    car3/doorL2/doorControlPart/openedDoor AT 1085 : BOOL := false;
    car3/doorL2/doorControlPart/closedDoor AT 1086 : BOOL := false;
    car3/doorL2/doorControlPart/lockedDoor AT 1087 : BOOL := false;
    car3/doorL2/doorControlPart/unlockedDoor AT 1088 : BOOL := false;
    car3/doorL2/doorControlPart/openingRequest AT 1089 : BOOL := false;
    car3/doorL2/doorControlPart/doorOpeningCmd AT 1090 : BOOL := false;
    car3/doorL2/doorControlPart/doorClosingCmd AT 1091 : BOOL := false;
    car3/doorL2/doorControlPart/doorLockingCmd AT 1083 : BOOL := false;
    car3/doorL2/doorControlPart/doorUnlockingCmd AT 1084 : BOOL := false;
    car3/doorL2/doorControlPart/closedDoorState AT 38 : BOOL := false;
    car3/doorL2/doorControlPart/openedDoorState AT 37 : BOOL := false;
    car3/doorL2/doorControlPart/faultState AT 533 : DINT := 0;
    car3/doorL2/doorControlPart/_X_10 AT 1103 : BOOL := true;
    car3/doorL2/doorControlPart/_X_11 AT 1104 : BOOL := false;
    car3/doorL2/doorControlPart/_X_12 AT 1105 : BOOL := false;
    car3/doorL2/doorControlPart/_X_13 AT 1106 : BOOL := false;
    car3/doorL2/doorControlPart/_X_14 AT 1107 : BOOL := false;
    car3/doorL2/doorControlPart/_X_15 AT 1108 : BOOL := false;
    car3/doorL2/doorControlPart/_X_16 AT 1109 : BOOL := false;
    car3/doorL2/door/compressedAir AT 115 : REAL := 200.0;
    car3/doorL2/door/cmdSupply AT 1016 : BOOL := true;
    car3/doorL2/door/sensorSupply AT 1015 : BOOL := true;
    car3/doorL2/door/openDoorCmd AT 1090 : BOOL := false;
    car3/doorL2/door/closeDoorCmd AT 1091 : BOOL := false;
    car3/doorL2/door/lockActive AT 1092 : BOOL := false;
    car3/doorL2/door/doorOpened AT 1085 : BOOL := false;
    car3/doorL2/door/doorClosed AT 1086 : BOOL := false;
    car3/doorL2/door/increment AT 121 : REAL := 0.0;
    car3/doorL2/door/openDoor AT 1116 : BOOL := false;
    car3/doorL2/door/closeDoor AT 1117 : BOOL := false;
    car3/doorL2/door/doorPosition AT 122 : REAL := 0.0;
    car3/doorL2/door/length AT 123 : REAL := 1000.0;
    car3/doorL2/door/doorClosedSensorLogic AT 1118 : BOOL := true;
    car3/doorL2/door/doorOpenedSensorLogic AT 1119 : BOOL := true;
    car3/doorL2/door/d_locking AT 1120 : BOOL := false;
    car3/doorL2/door/v_d_locking AT 124 : REAL := 50.0;
    car3/doorL2/door/d_doorClosedSensor AT 1121 : BOOL := false;
    car3/doorL2/door/v_d_doorClosedSensor AT 1122 : BOOL := false;
    car3/doorL2/door/d_doorOpenedSensor AT 1123 : BOOL := false;
    car3/doorL2/door/v_d_doorOpenedSensor AT 1124 : BOOL := false;
    car3/doorL3/compressedAir AT 114 : REAL := 200.0;
    car3/doorL3/cmdSupply AT 1014 : BOOL := true;
    car3/doorL3/sensorSupply AT 1013 : BOOL := true;
    car3/doorL3/enableOpening AT 1019 : BOOL := false;
    car3/doorL3/enableClosing AT 1020 : BOOL := false;
    car3/doorL3/closedDoorState AT 36 : BOOL := false;
    car3/doorL3/openedDoorState AT 35 : BOOL := false;
    car3/doorL3/faultState AT 532 : DINT := 0;
    car3/doorL3/doorPB/doorPB AT 1131 : BOOL := false;
    car3/doorL3/doorPB/button AT 1135 : BOOL := false;
    car3/doorL3/doorPB/_X_10 AT 1136 : BOOL := true;
    car3/doorL3/doorPB/_X_11 AT 1137 : BOOL := false;
    car3/doorL3/doorPB/_X_12 AT 1138 : BOOL := false;
    car3/doorL3/doorLocking/lockingCmd AT 1125 : BOOL := false;
    car3/doorL3/doorLocking/unlockingCmd AT 1126 : BOOL := false;
    car3/doorL3/doorLocking/doorLocked AT 1129 : BOOL := false;
    car3/doorL3/doorLocking/doorUnlocked AT 1130 : BOOL := false;
    car3/doorL3/doorLocking/lockActive AT 1134 : BOOL := false;
    car3/doorL3/doorLocking/i_rs1 AT 662 : DINT := 0;
    car3/doorL3/doorLocking/d_unlockedSensor AT 1140 : BOOL := false;
    car3/doorL3/doorLocking/v_d_unlockedSensor AT 1141 : BOOL := false;
    car3/doorL3/doorLocking/d_lockedSensor AT 1142 : BOOL := false;
    car3/doorL3/doorLocking/v_d_lockedSensor AT 1143 : BOOL := false;
    car3/doorL3/doorControlPart/enableOpening AT 1019 : BOOL := false;
    car3/doorL3/doorControlPart/enableClosing AT 1020 : BOOL := false;
    car3/doorL3/doorControlPart/openedDoor AT 1127 : BOOL := false;
    car3/doorL3/doorControlPart/closedDoor AT 1128 : BOOL := false;
    car3/doorL3/doorControlPart/lockedDoor AT 1129 : BOOL := false;
    car3/doorL3/doorControlPart/unlockedDoor AT 1130 : BOOL := false;
    car3/doorL3/doorControlPart/openingRequest AT 1131 : BOOL := false;
    car3/doorL3/doorControlPart/doorOpeningCmd AT 1132 : BOOL := false;
    car3/doorL3/doorControlPart/doorClosingCmd AT 1133 : BOOL := false;
    car3/doorL3/doorControlPart/doorLockingCmd AT 1125 : BOOL := false;
    car3/doorL3/doorControlPart/doorUnlockingCmd AT 1126 : BOOL := false;
    car3/doorL3/doorControlPart/closedDoorState AT 36 : BOOL := false;
    car3/doorL3/doorControlPart/openedDoorState AT 35 : BOOL := false;
    car3/doorL3/doorControlPart/faultState AT 532 : DINT := 0;
    car3/doorL3/doorControlPart/_X_10 AT 1145 : BOOL := true;
    car3/doorL3/doorControlPart/_X_11 AT 1146 : BOOL := false;
    car3/doorL3/doorControlPart/_X_12 AT 1147 : BOOL := false;
    car3/doorL3/doorControlPart/_X_13 AT 1148 : BOOL := false;
    car3/doorL3/doorControlPart/_X_14 AT 1149 : BOOL := false;
    car3/doorL3/doorControlPart/_X_15 AT 1150 : BOOL := false;
    car3/doorL3/doorControlPart/_X_16 AT 1151 : BOOL := false;
    car3/doorL3/door/compressedAir AT 114 : REAL := 200.0;
    car3/doorL3/door/cmdSupply AT 1014 : BOOL := true;
    car3/doorL3/door/sensorSupply AT 1013 : BOOL := true;
    car3/doorL3/door/openDoorCmd AT 1132 : BOOL := false;
    car3/doorL3/door/closeDoorCmd AT 1133 : BOOL := false;
    car3/doorL3/door/lockActive AT 1134 : BOOL := false;
    car3/doorL3/door/doorOpened AT 1127 : BOOL := false;
    car3/doorL3/door/doorClosed AT 1128 : BOOL := false;
    car3/doorL3/door/increment AT 125 : REAL := 0.0;
    car3/doorL3/door/openDoor AT 1158 : BOOL := false;
    car3/doorL3/door/closeDoor AT 1159 : BOOL := false;
    car3/doorL3/door/doorPosition AT 126 : REAL := 0.0;
    car3/doorL3/door/length AT 127 : REAL := 1000.0;
    car3/doorL3/door/doorClosedSensorLogic AT 1160 : BOOL := true;
    car3/doorL3/door/doorOpenedSensorLogic AT 1161 : BOOL := true;
    car3/doorL3/door/d_locking AT 1162 : BOOL := false;
    car3/doorL3/door/v_d_locking AT 128 : REAL := 50.0;
    car3/doorL3/door/d_doorClosedSensor AT 1163 : BOOL := false;
    car3/doorL3/door/v_d_doorClosedSensor AT 1164 : BOOL := false;
    car3/doorL3/door/d_doorOpenedSensor AT 1165 : BOOL := false;
    car3/doorL3/door/v_d_doorOpenedSensor AT 1166 : BOOL := false;
    car3/doorR1/compressedAir AT 113 : REAL := 200.0;
    car3/doorR1/cmdSupply AT 1012 : BOOL := true;
    car3/doorR1/sensorSupply AT 1011 : BOOL := true;
    car3/doorR1/enableOpening AT 1021 : BOOL := false;
    car3/doorR1/enableClosing AT 1022 : BOOL := false;
    car3/doorR1/closedDoorState AT 34 : BOOL := false;
    car3/doorR1/openedDoorState AT 33 : BOOL := false;
    car3/doorR1/faultState AT 531 : DINT := 0;
    car3/doorR1/doorPB/doorPB AT 1173 : BOOL := false;
    car3/doorR1/doorPB/button AT 1177 : BOOL := false;
    car3/doorR1/doorPB/_X_10 AT 1178 : BOOL := true;
    car3/doorR1/doorPB/_X_11 AT 1179 : BOOL := false;
    car3/doorR1/doorPB/_X_12 AT 1180 : BOOL := false;
    car3/doorR1/doorLocking/lockingCmd AT 1167 : BOOL := false;
    car3/doorR1/doorLocking/unlockingCmd AT 1168 : BOOL := false;
    car3/doorR1/doorLocking/doorLocked AT 1171 : BOOL := false;
    car3/doorR1/doorLocking/doorUnlocked AT 1172 : BOOL := false;
    car3/doorR1/doorLocking/lockActive AT 1176 : BOOL := false;
    car3/doorR1/doorLocking/i_rs1 AT 665 : DINT := 0;
    car3/doorR1/doorLocking/d_unlockedSensor AT 1182 : BOOL := false;
    car3/doorR1/doorLocking/v_d_unlockedSensor AT 1183 : BOOL := false;
    car3/doorR1/doorLocking/d_lockedSensor AT 1184 : BOOL := false;
    car3/doorR1/doorLocking/v_d_lockedSensor AT 1185 : BOOL := false;
    car3/doorR1/doorControlPart/enableOpening AT 1021 : BOOL := false;
    car3/doorR1/doorControlPart/enableClosing AT 1022 : BOOL := false;
    car3/doorR1/doorControlPart/openedDoor AT 1169 : BOOL := false;
    car3/doorR1/doorControlPart/closedDoor AT 1170 : BOOL := false;
    car3/doorR1/doorControlPart/lockedDoor AT 1171 : BOOL := false;
    car3/doorR1/doorControlPart/unlockedDoor AT 1172 : BOOL := false;
    car3/doorR1/doorControlPart/openingRequest AT 1173 : BOOL := false;
    car3/doorR1/doorControlPart/doorOpeningCmd AT 1174 : BOOL := false;
    car3/doorR1/doorControlPart/doorClosingCmd AT 1175 : BOOL := false;
    car3/doorR1/doorControlPart/doorLockingCmd AT 1167 : BOOL := false;
    car3/doorR1/doorControlPart/doorUnlockingCmd AT 1168 : BOOL := false;
    car3/doorR1/doorControlPart/closedDoorState AT 34 : BOOL := false;
    car3/doorR1/doorControlPart/openedDoorState AT 33 : BOOL := false;
    car3/doorR1/doorControlPart/faultState AT 531 : DINT := 0;
    car3/doorR1/doorControlPart/_X_10 AT 1187 : BOOL := true;
    car3/doorR1/doorControlPart/_X_11 AT 1188 : BOOL := false;
    car3/doorR1/doorControlPart/_X_12 AT 1189 : BOOL := false;
    car3/doorR1/doorControlPart/_X_13 AT 1190 : BOOL := false;
    car3/doorR1/doorControlPart/_X_14 AT 1191 : BOOL := false;
    car3/doorR1/doorControlPart/_X_15 AT 1192 : BOOL := false;
    car3/doorR1/doorControlPart/_X_16 AT 1193 : BOOL := false;
    car3/doorR1/door/compressedAir AT 113 : REAL := 200.0;
    car3/doorR1/door/cmdSupply AT 1012 : BOOL := true;
    car3/doorR1/door/sensorSupply AT 1011 : BOOL := true;
    car3/doorR1/door/openDoorCmd AT 1174 : BOOL := false;
    car3/doorR1/door/closeDoorCmd AT 1175 : BOOL := false;
    car3/doorR1/door/lockActive AT 1176 : BOOL := false;
    car3/doorR1/door/doorOpened AT 1169 : BOOL := false;
    car3/doorR1/door/doorClosed AT 1170 : BOOL := false;
    car3/doorR1/door/increment AT 129 : REAL := 0.0;
    car3/doorR1/door/openDoor AT 1200 : BOOL := false;
    car3/doorR1/door/closeDoor AT 1201 : BOOL := false;
    car3/doorR1/door/doorPosition AT 130 : REAL := 0.0;
    car3/doorR1/door/length AT 131 : REAL := 1000.0;
    car3/doorR1/door/doorClosedSensorLogic AT 1202 : BOOL := true;
    car3/doorR1/door/doorOpenedSensorLogic AT 1203 : BOOL := true;
    car3/doorR1/door/d_locking AT 1204 : BOOL := false;
    car3/doorR1/door/v_d_locking AT 132 : REAL := 50.0;
    car3/doorR1/door/d_doorClosedSensor AT 1205 : BOOL := false;
    car3/doorR1/door/v_d_doorClosedSensor AT 1206 : BOOL := false;
    car3/doorR1/door/d_doorOpenedSensor AT 1207 : BOOL := false;
    car3/doorR1/door/v_d_doorOpenedSensor AT 1208 : BOOL := false;
    car3/doorR2/compressedAir AT 112 : REAL := 200.0;
    car3/doorR2/cmdSupply AT 1010 : BOOL := true;
    car3/doorR2/sensorSupply AT 1009 : BOOL := true;
    car3/doorR2/enableOpening AT 1021 : BOOL := false;
    car3/doorR2/enableClosing AT 1022 : BOOL := false;
    car3/doorR2/closedDoorState AT 32 : BOOL := false;
    car3/doorR2/openedDoorState AT 31 : BOOL := false;
    car3/doorR2/faultState AT 530 : DINT := 0;
    car3/doorR2/doorPB/doorPB AT 1215 : BOOL := false;
    car3/doorR2/doorPB/button AT 1219 : BOOL := false;
    car3/doorR2/doorPB/_X_10 AT 1220 : BOOL := true;
    car3/doorR2/doorPB/_X_11 AT 1221 : BOOL := false;
    car3/doorR2/doorPB/_X_12 AT 1222 : BOOL := false;
    car3/doorR2/doorLocking/lockingCmd AT 1209 : BOOL := false;
    car3/doorR2/doorLocking/unlockingCmd AT 1210 : BOOL := false;
    car3/doorR2/doorLocking/doorLocked AT 1213 : BOOL := false;
    car3/doorR2/doorLocking/doorUnlocked AT 1214 : BOOL := false;
    car3/doorR2/doorLocking/lockActive AT 1218 : BOOL := false;
    car3/doorR2/doorLocking/i_rs1 AT 668 : DINT := 0;
    car3/doorR2/doorLocking/d_unlockedSensor AT 1224 : BOOL := false;
    car3/doorR2/doorLocking/v_d_unlockedSensor AT 1225 : BOOL := false;
    car3/doorR2/doorLocking/d_lockedSensor AT 1226 : BOOL := false;
    car3/doorR2/doorLocking/v_d_lockedSensor AT 1227 : BOOL := false;
    car3/doorR2/doorControlPart/enableOpening AT 1021 : BOOL := false;
    car3/doorR2/doorControlPart/enableClosing AT 1022 : BOOL := false;
    car3/doorR2/doorControlPart/openedDoor AT 1211 : BOOL := false;
    car3/doorR2/doorControlPart/closedDoor AT 1212 : BOOL := false;
    car3/doorR2/doorControlPart/lockedDoor AT 1213 : BOOL := false;
    car3/doorR2/doorControlPart/unlockedDoor AT 1214 : BOOL := false;
    car3/doorR2/doorControlPart/openingRequest AT 1215 : BOOL := false;
    car3/doorR2/doorControlPart/doorOpeningCmd AT 1216 : BOOL := false;
    car3/doorR2/doorControlPart/doorClosingCmd AT 1217 : BOOL := false;
    car3/doorR2/doorControlPart/doorLockingCmd AT 1209 : BOOL := false;
    car3/doorR2/doorControlPart/doorUnlockingCmd AT 1210 : BOOL := false;
    car3/doorR2/doorControlPart/closedDoorState AT 32 : BOOL := false;
    car3/doorR2/doorControlPart/openedDoorState AT 31 : BOOL := false;
    car3/doorR2/doorControlPart/faultState AT 530 : DINT := 0;
    car3/doorR2/doorControlPart/_X_10 AT 1229 : BOOL := true;
    car3/doorR2/doorControlPart/_X_11 AT 1230 : BOOL := false;
    car3/doorR2/doorControlPart/_X_12 AT 1231 : BOOL := false;
    car3/doorR2/doorControlPart/_X_13 AT 1232 : BOOL := false;
    car3/doorR2/doorControlPart/_X_14 AT 1233 : BOOL := false;
    car3/doorR2/doorControlPart/_X_15 AT 1234 : BOOL := false;
    car3/doorR2/doorControlPart/_X_16 AT 1235 : BOOL := false;
    car3/doorR2/door/compressedAir AT 112 : REAL := 200.0;
    car3/doorR2/door/cmdSupply AT 1010 : BOOL := true;
    car3/doorR2/door/sensorSupply AT 1009 : BOOL := true;
    car3/doorR2/door/openDoorCmd AT 1216 : BOOL := false;
    car3/doorR2/door/closeDoorCmd AT 1217 : BOOL := false;
    car3/doorR2/door/lockActive AT 1218 : BOOL := false;
    car3/doorR2/door/doorOpened AT 1211 : BOOL := false;
    car3/doorR2/door/doorClosed AT 1212 : BOOL := false;
    car3/doorR2/door/increment AT 133 : REAL := 0.0;
    car3/doorR2/door/openDoor AT 1242 : BOOL := false;
    car3/doorR2/door/closeDoor AT 1243 : BOOL := false;
    car3/doorR2/door/doorPosition AT 134 : REAL := 0.0;
    car3/doorR2/door/length AT 135 : REAL := 1000.0;
    car3/doorR2/door/doorClosedSensorLogic AT 1244 : BOOL := true;
    car3/doorR2/door/doorOpenedSensorLogic AT 1245 : BOOL := true;
    car3/doorR2/door/d_locking AT 1246 : BOOL := false;
    car3/doorR2/door/v_d_locking AT 136 : REAL := 50.0;
    car3/doorR2/door/d_doorClosedSensor AT 1247 : BOOL := false;
    car3/doorR2/door/v_d_doorClosedSensor AT 1248 : BOOL := false;
    car3/doorR2/door/d_doorOpenedSensor AT 1249 : BOOL := false;
    car3/doorR2/door/v_d_doorOpenedSensor AT 1250 : BOOL := false;
    car3/doorR3/compressedAir AT 111 : REAL := 200.0;
    car3/doorR3/cmdSupply AT 1008 : BOOL := true;
    car3/doorR3/sensorSupply AT 1007 : BOOL := true;
    car3/doorR3/enableOpening AT 1021 : BOOL := false;
    car3/doorR3/enableClosing AT 1022 : BOOL := false;
    car3/doorR3/closedDoorState AT 30 : BOOL := false;
    car3/doorR3/openedDoorState AT 29 : BOOL := false;
    car3/doorR3/faultState AT 529 : DINT := 0;
    car3/doorR3/doorPB/doorPB AT 1257 : BOOL := false;
    car3/doorR3/doorPB/button AT 1261 : BOOL := false;
    car3/doorR3/doorPB/_X_10 AT 1262 : BOOL := true;
    car3/doorR3/doorPB/_X_11 AT 1263 : BOOL := false;
    car3/doorR3/doorPB/_X_12 AT 1264 : BOOL := false;
    car3/doorR3/doorLocking/lockingCmd AT 1251 : BOOL := false;
    car3/doorR3/doorLocking/unlockingCmd AT 1252 : BOOL := false;
    car3/doorR3/doorLocking/doorLocked AT 1255 : BOOL := false;
    car3/doorR3/doorLocking/doorUnlocked AT 1256 : BOOL := false;
    car3/doorR3/doorLocking/lockActive AT 1260 : BOOL := false;
    car3/doorR3/doorLocking/i_rs1 AT 671 : DINT := 0;
    car3/doorR3/doorLocking/d_unlockedSensor AT 1266 : BOOL := false;
    car3/doorR3/doorLocking/v_d_unlockedSensor AT 1267 : BOOL := false;
    car3/doorR3/doorLocking/d_lockedSensor AT 1268 : BOOL := false;
    car3/doorR3/doorLocking/v_d_lockedSensor AT 1269 : BOOL := false;
    car3/doorR3/doorControlPart/enableOpening AT 1021 : BOOL := false;
    car3/doorR3/doorControlPart/enableClosing AT 1022 : BOOL := false;
    car3/doorR3/doorControlPart/openedDoor AT 1253 : BOOL := false;
    car3/doorR3/doorControlPart/closedDoor AT 1254 : BOOL := false;
    car3/doorR3/doorControlPart/lockedDoor AT 1255 : BOOL := false;
    car3/doorR3/doorControlPart/unlockedDoor AT 1256 : BOOL := false;
    car3/doorR3/doorControlPart/openingRequest AT 1257 : BOOL := false;
    car3/doorR3/doorControlPart/doorOpeningCmd AT 1258 : BOOL := false;
    car3/doorR3/doorControlPart/doorClosingCmd AT 1259 : BOOL := false;
    car3/doorR3/doorControlPart/doorLockingCmd AT 1251 : BOOL := false;
    car3/doorR3/doorControlPart/doorUnlockingCmd AT 1252 : BOOL := false;
    car3/doorR3/doorControlPart/closedDoorState AT 30 : BOOL := false;
    car3/doorR3/doorControlPart/openedDoorState AT 29 : BOOL := false;
    car3/doorR3/doorControlPart/faultState AT 529 : DINT := 0;
    car3/doorR3/doorControlPart/_X_10 AT 1271 : BOOL := true;
    car3/doorR3/doorControlPart/_X_11 AT 1272 : BOOL := false;
    car3/doorR3/doorControlPart/_X_12 AT 1273 : BOOL := false;
    car3/doorR3/doorControlPart/_X_13 AT 1274 : BOOL := false;
    car3/doorR3/doorControlPart/_X_14 AT 1275 : BOOL := false;
    car3/doorR3/doorControlPart/_X_15 AT 1276 : BOOL := false;
    car3/doorR3/doorControlPart/_X_16 AT 1277 : BOOL := false;
    car3/doorR3/door/compressedAir AT 111 : REAL := 200.0;
    car3/doorR3/door/cmdSupply AT 1008 : BOOL := true;
    car3/doorR3/door/sensorSupply AT 1007 : BOOL := true;
    car3/doorR3/door/openDoorCmd AT 1258 : BOOL := false;
    car3/doorR3/door/closeDoorCmd AT 1259 : BOOL := false;
    car3/doorR3/door/lockActive AT 1260 : BOOL := false;
    car3/doorR3/door/doorOpened AT 1253 : BOOL := false;
    car3/doorR3/door/doorClosed AT 1254 : BOOL := false;
    car3/doorR3/door/increment AT 137 : REAL := 0.0;
    car3/doorR3/door/openDoor AT 1284 : BOOL := false;
    car3/doorR3/door/closeDoor AT 1285 : BOOL := false;
    car3/doorR3/door/doorPosition AT 138 : REAL := 0.0;
    car3/doorR3/door/length AT 139 : REAL := 1000.0;
    car3/doorR3/door/doorClosedSensorLogic AT 1286 : BOOL := true;
    car3/doorR3/door/doorOpenedSensorLogic AT 1287 : BOOL := true;
    car3/doorR3/door/d_locking AT 1288 : BOOL := false;
    car3/doorR3/door/v_d_locking AT 140 : REAL := 50.0;
    car3/doorR3/door/d_doorClosedSensor AT 1289 : BOOL := false;
    car3/doorR3/door/v_d_doorClosedSensor AT 1290 : BOOL := false;
    car3/doorR3/door/d_doorOpenedSensor AT 1291 : BOOL := false;
    car3/doorR3/door/v_d_doorOpenedSensor AT 1292 : BOOL := false;
    motorCar2/AuthorizationClosingLeftC1 AT 101 : BOOL := false;
    motorCar2/AuthorizationOpeningRightC1 AT 102 : BOOL := false;
    motorCar2/AuthorizationClosingRightC1 AT 103 : BOOL := false;
    motorCar2/AuthorizationOpeningLeftC1 AT 104 : BOOL := false;
    motorCar2/AuthorizationClosingLeftC2 AT 105 : BOOL := false;
    motorCar2/AuthorizationOpeningRightC2 AT 106 : BOOL := false;
    motorCar2/AuthorizationClosingRightC2 AT 107 : BOOL := false;
    motorCar2/AuthorizationOpeningLeftC2 AT 108 : BOOL := false;
    motorCar2/doorL1Closed AT 22 : BOOL := false;
    motorCar2/doorL1Opened AT 21 : BOOL := false;
    motorCar2/doorL1Fault AT 528 : DINT := 0;
    motorCar2/doorL2Closed AT 20 : BOOL := false;
    motorCar2/doorL2Opened AT 19 : BOOL := false;
    motorCar2/doorL2Fault AT 527 : DINT := 0;
    motorCar2/doorL3Closed AT 18 : BOOL := false;
    motorCar2/doorL3Opened AT 17 : BOOL := false;
    motorCar2/doorL3Fault AT 526 : DINT := 0;
    motorCar2/doorR1Closed AT 16 : BOOL := false;
    motorCar2/doorR1Opened AT 15 : BOOL := false;
    motorCar2/doorR1Fault AT 525 : DINT := 0;
    motorCar2/doorR2Closed AT 14 : BOOL := false;
    motorCar2/doorR2Opened AT 13 : BOOL := false;
    motorCar2/doorR2Fault AT 524 : DINT := 0;
    motorCar2/doorR3Closed AT 12 : BOOL := false;
    motorCar2/doorR3Opened AT 11 : BOOL := false;
    motorCar2/doorR3Fault AT 523 : DINT := 0;
    motorCar2/AlarmD1L AT 10 : BOOL := false;
    motorCar2/AlarmD2L AT 9 : BOOL := false;
    motorCar2/AlarmD3L AT 8 : BOOL := false;
    motorCar2/AlarmD1R AT 7 : BOOL := false;
    motorCar2/AlarmD2R AT 6 : BOOL := false;
    motorCar2/AlarmD3R AT 5 : BOOL := false;
    motorCar2/authorizations/AuthorizationClosingLeftC1 AT 101 : BOOL := false;
    motorCar2/authorizations/AuthorizationOpeningRightC1 AT 102 : BOOL := false;
    motorCar2/authorizations/AuthorizationClosingRightC1 AT 103 : BOOL := false;
    motorCar2/authorizations/AuthorizationOpeningLeftC1 AT 104 : BOOL := false;
    motorCar2/authorizations/AuthorizationClosingLeftC2 AT 105 : BOOL := false;
    motorCar2/authorizations/AuthorizationOpeningRightC2 AT 106 : BOOL := false;
    motorCar2/authorizations/AuthorizationClosingRightC2 AT 107 : BOOL := false;
    motorCar2/authorizations/AuthorizationOpeningLeftC2 AT 108 : BOOL := false;
    motorCar2/authorizations/AuthorizationOpeningLeft AT 1305 : BOOL := false;
    motorCar2/authorizations/AuthorizationClosingLeft AT 1306 : BOOL := false;
    motorCar2/authorizations/AuthorizationOpeningRight AT 1307 : BOOL := false;
    motorCar2/authorizations/AuthorizationClosingRight AT 1308 : BOOL := false;
    motorCar2/alarms/AlarmD1L AT 10 : BOOL := false;
    motorCar2/alarms/AlarmD2L AT 9 : BOOL := false;
    motorCar2/alarms/AlarmD3L AT 8 : BOOL := false;
    motorCar2/alarms/AlarmD1R AT 7 : BOOL := false;
    motorCar2/alarms/AlarmD2R AT 6 : BOOL := false;
    motorCar2/alarms/AlarmD3R AT 5 : BOOL := false;
    motorCar2/alarms/AlarmD1L/enableAlarm AT 1320 : BOOL := false;
    motorCar2/alarms/AlarmD1L/resetKey AT 1319 : BOOL := false;
    motorCar2/alarms/AlarmD1L/alarm AT 10 : BOOL := false;
    motorCar2/alarms/AlarmD1L/i_rs1 AT 673 : DINT := 0;
    motorCar2/alarms/AlarmD2L/enableAlarm AT 1318 : BOOL := false;
    motorCar2/alarms/AlarmD2L/resetKey AT 1317 : BOOL := false;
    motorCar2/alarms/AlarmD2L/alarm AT 9 : BOOL := false;
    motorCar2/alarms/AlarmD2L/i_rs1 AT 675 : DINT := 0;
    motorCar2/alarms/AlarmD3L/enableAlarm AT 1316 : BOOL := false;
    motorCar2/alarms/AlarmD3L/resetKey AT 1315 : BOOL := false;
    motorCar2/alarms/AlarmD3L/alarm AT 8 : BOOL := false;
    motorCar2/alarms/AlarmD3L/i_rs1 AT 677 : DINT := 0;
    motorCar2/alarms/AlarmD1R/enableAlarm AT 1314 : BOOL := false;
    motorCar2/alarms/AlarmD1R/resetKey AT 1313 : BOOL := false;
    motorCar2/alarms/AlarmD1R/alarm AT 7 : BOOL := false;
    motorCar2/alarms/AlarmD1R/i_rs1 AT 679 : DINT := 0;
    motorCar2/alarms/AlarmD2R/enableAlarm AT 1312 : BOOL := false;
    motorCar2/alarms/AlarmD2R/resetKey AT 1311 : BOOL := false;
    motorCar2/alarms/AlarmD2R/alarm AT 6 : BOOL := false;
    motorCar2/alarms/AlarmD2R/i_rs1 AT 681 : DINT := 0;
    motorCar2/alarms/AlarmD3R/enableAlarm AT 1310 : BOOL := false;
    motorCar2/alarms/AlarmD3R/resetKey AT 1309 : BOOL := false;
    motorCar2/alarms/AlarmD3R/alarm AT 5 : BOOL := false;
    motorCar2/alarms/AlarmD3R/i_rs1 AT 683 : DINT := 0;
    motorCar2/doorL1/compressedAir AT 146 : REAL := 200.0;
    motorCar2/doorL1/cmdSupply AT 1304 : BOOL := true;
    motorCar2/doorL1/sensorSupply AT 1303 : BOOL := true;
    motorCar2/doorL1/enableOpening AT 1305 : BOOL := false;
    motorCar2/doorL1/enableClosing AT 1306 : BOOL := false;
    motorCar2/doorL1/closedDoorState AT 22 : BOOL := false;
    motorCar2/doorL1/openedDoorState AT 21 : BOOL := false;
    motorCar2/doorL1/faultState AT 528 : DINT := 0;
    motorCar2/doorL1/doorPB/doorPB AT 1333 : BOOL := false;
    motorCar2/doorL1/doorPB/button AT 1337 : BOOL := false;
    motorCar2/doorL1/doorPB/_X_10 AT 1338 : BOOL := true;
    motorCar2/doorL1/doorPB/_X_11 AT 1339 : BOOL := false;
    motorCar2/doorL1/doorPB/_X_12 AT 1340 : BOOL := false;
    motorCar2/doorL1/doorLocking/lockingCmd AT 1327 : BOOL := false;
    motorCar2/doorL1/doorLocking/unlockingCmd AT 1328 : BOOL := false;
    motorCar2/doorL1/doorLocking/doorLocked AT 1331 : BOOL := false;
    motorCar2/doorL1/doorLocking/doorUnlocked AT 1332 : BOOL := false;
    motorCar2/doorL1/doorLocking/lockActive AT 1336 : BOOL := false;
    motorCar2/doorL1/doorLocking/i_rs1 AT 686 : DINT := 0;
    motorCar2/doorL1/doorLocking/d_unlockedSensor AT 1342 : BOOL := false;
    motorCar2/doorL1/doorLocking/v_d_unlockedSensor AT 1343 : BOOL := false;
    motorCar2/doorL1/doorLocking/d_lockedSensor AT 1344 : BOOL := false;
    motorCar2/doorL1/doorLocking/v_d_lockedSensor AT 1345 : BOOL := false;
    motorCar2/doorL1/doorControlPart/enableOpening AT 1305 : BOOL := false;
    motorCar2/doorL1/doorControlPart/enableClosing AT 1306 : BOOL := false;
    motorCar2/doorL1/doorControlPart/openedDoor AT 1329 : BOOL := false;
    motorCar2/doorL1/doorControlPart/closedDoor AT 1330 : BOOL := false;
    motorCar2/doorL1/doorControlPart/lockedDoor AT 1331 : BOOL := false;
    motorCar2/doorL1/doorControlPart/unlockedDoor AT 1332 : BOOL := false;
    motorCar2/doorL1/doorControlPart/openingRequest AT 1333 : BOOL := false;
    motorCar2/doorL1/doorControlPart/doorOpeningCmd AT 1334 : BOOL := false;
    motorCar2/doorL1/doorControlPart/doorClosingCmd AT 1335 : BOOL := false;
    motorCar2/doorL1/doorControlPart/doorLockingCmd AT 1327 : BOOL := false;
    motorCar2/doorL1/doorControlPart/doorUnlockingCmd AT 1328 : BOOL := false;
    motorCar2/doorL1/doorControlPart/closedDoorState AT 22 : BOOL := false;
    motorCar2/doorL1/doorControlPart/openedDoorState AT 21 : BOOL := false;
    motorCar2/doorL1/doorControlPart/faultState AT 528 : DINT := 0;
    motorCar2/doorL1/doorControlPart/_X_10 AT 1347 : BOOL := true;
    motorCar2/doorL1/doorControlPart/_X_11 AT 1348 : BOOL := false;
    motorCar2/doorL1/doorControlPart/_X_12 AT 1349 : BOOL := false;
    motorCar2/doorL1/doorControlPart/_X_13 AT 1350 : BOOL := false;
    motorCar2/doorL1/doorControlPart/_X_14 AT 1351 : BOOL := false;
    motorCar2/doorL1/doorControlPart/_X_15 AT 1352 : BOOL := false;
    motorCar2/doorL1/doorControlPart/_X_16 AT 1353 : BOOL := false;
    motorCar2/doorL1/door/compressedAir AT 146 : REAL := 200.0;
    motorCar2/doorL1/door/cmdSupply AT 1304 : BOOL := true;
    motorCar2/doorL1/door/sensorSupply AT 1303 : BOOL := true;
    motorCar2/doorL1/door/openDoorCmd AT 1334 : BOOL := false;
    motorCar2/doorL1/door/closeDoorCmd AT 1335 : BOOL := false;
    motorCar2/doorL1/door/lockActive AT 1336 : BOOL := false;
    motorCar2/doorL1/door/doorOpened AT 1329 : BOOL := false;
    motorCar2/doorL1/door/doorClosed AT 1330 : BOOL := false;
    motorCar2/doorL1/door/increment AT 147 : REAL := 0.0;
    motorCar2/doorL1/door/openDoor AT 1360 : BOOL := false;
    motorCar2/doorL1/door/closeDoor AT 1361 : BOOL := false;
    motorCar2/doorL1/door/doorPosition AT 148 : REAL := 0.0;
    motorCar2/doorL1/door/length AT 149 : REAL := 1000.0;
    motorCar2/doorL1/door/doorClosedSensorLogic AT 1362 : BOOL := true;
    motorCar2/doorL1/door/doorOpenedSensorLogic AT 1363 : BOOL := true;
    motorCar2/doorL1/door/d_locking AT 1364 : BOOL := false;
    motorCar2/doorL1/door/v_d_locking AT 150 : REAL := 50.0;
    motorCar2/doorL1/door/d_doorClosedSensor AT 1365 : BOOL := false;
    motorCar2/doorL1/door/v_d_doorClosedSensor AT 1366 : BOOL := false;
    motorCar2/doorL1/door/d_doorOpenedSensor AT 1367 : BOOL := false;
    motorCar2/doorL1/door/v_d_doorOpenedSensor AT 1368 : BOOL := false;
    motorCar2/doorL2/compressedAir AT 145 : REAL := 200.0;
    motorCar2/doorL2/cmdSupply AT 1302 : BOOL := true;
    motorCar2/doorL2/sensorSupply AT 1301 : BOOL := true;
    motorCar2/doorL2/enableOpening AT 1305 : BOOL := false;
    motorCar2/doorL2/enableClosing AT 1306 : BOOL := false;
    motorCar2/doorL2/closedDoorState AT 20 : BOOL := false;
    motorCar2/doorL2/openedDoorState AT 19 : BOOL := false;
    motorCar2/doorL2/faultState AT 527 : DINT := 0;
    motorCar2/doorL2/doorPB/doorPB AT 1375 : BOOL := false;
    motorCar2/doorL2/doorPB/button AT 1379 : BOOL := false;
    motorCar2/doorL2/doorPB/_X_10 AT 1380 : BOOL := true;
    motorCar2/doorL2/doorPB/_X_11 AT 1381 : BOOL := false;
    motorCar2/doorL2/doorPB/_X_12 AT 1382 : BOOL := false;
    motorCar2/doorL2/doorLocking/lockingCmd AT 1369 : BOOL := false;
    motorCar2/doorL2/doorLocking/unlockingCmd AT 1370 : BOOL := false;
    motorCar2/doorL2/doorLocking/doorLocked AT 1373 : BOOL := false;
    motorCar2/doorL2/doorLocking/doorUnlocked AT 1374 : BOOL := false;
    motorCar2/doorL2/doorLocking/lockActive AT 1378 : BOOL := false;
    motorCar2/doorL2/doorLocking/i_rs1 AT 689 : DINT := 0;
    motorCar2/doorL2/doorLocking/d_unlockedSensor AT 1384 : BOOL := false;
    motorCar2/doorL2/doorLocking/v_d_unlockedSensor AT 1385 : BOOL := false;
    motorCar2/doorL2/doorLocking/d_lockedSensor AT 1386 : BOOL := false;
    motorCar2/doorL2/doorLocking/v_d_lockedSensor AT 1387 : BOOL := false;
    motorCar2/doorL2/doorControlPart/enableOpening AT 1305 : BOOL := false;
    motorCar2/doorL2/doorControlPart/enableClosing AT 1306 : BOOL := false;
    motorCar2/doorL2/doorControlPart/openedDoor AT 1371 : BOOL := false;
    motorCar2/doorL2/doorControlPart/closedDoor AT 1372 : BOOL := false;
    motorCar2/doorL2/doorControlPart/lockedDoor AT 1373 : BOOL := false;
    motorCar2/doorL2/doorControlPart/unlockedDoor AT 1374 : BOOL := false;
    motorCar2/doorL2/doorControlPart/openingRequest AT 1375 : BOOL := false;
    motorCar2/doorL2/doorControlPart/doorOpeningCmd AT 1376 : BOOL := false;
    motorCar2/doorL2/doorControlPart/doorClosingCmd AT 1377 : BOOL := false;
    motorCar2/doorL2/doorControlPart/doorLockingCmd AT 1369 : BOOL := false;
    motorCar2/doorL2/doorControlPart/doorUnlockingCmd AT 1370 : BOOL := false;
    motorCar2/doorL2/doorControlPart/closedDoorState AT 20 : BOOL := false;
    motorCar2/doorL2/doorControlPart/openedDoorState AT 19 : BOOL := false;
    motorCar2/doorL2/doorControlPart/faultState AT 527 : DINT := 0;
    motorCar2/doorL2/doorControlPart/_X_10 AT 1389 : BOOL := true;
    motorCar2/doorL2/doorControlPart/_X_11 AT 1390 : BOOL := false;
    motorCar2/doorL2/doorControlPart/_X_12 AT 1391 : BOOL := false;
    motorCar2/doorL2/doorControlPart/_X_13 AT 1392 : BOOL := false;
    motorCar2/doorL2/doorControlPart/_X_14 AT 1393 : BOOL := false;
    motorCar2/doorL2/doorControlPart/_X_15 AT 1394 : BOOL := false;
    motorCar2/doorL2/doorControlPart/_X_16 AT 1395 : BOOL := false;
    motorCar2/doorL2/door/compressedAir AT 145 : REAL := 200.0;
    motorCar2/doorL2/door/cmdSupply AT 1302 : BOOL := true;
    motorCar2/doorL2/door/sensorSupply AT 1301 : BOOL := true;
    motorCar2/doorL2/door/openDoorCmd AT 1376 : BOOL := false;
    motorCar2/doorL2/door/closeDoorCmd AT 1377 : BOOL := false;
    motorCar2/doorL2/door/lockActive AT 1378 : BOOL := false;
    motorCar2/doorL2/door/doorOpened AT 1371 : BOOL := false;
    motorCar2/doorL2/door/doorClosed AT 1372 : BOOL := false;
    motorCar2/doorL2/door/increment AT 151 : REAL := 0.0;
    motorCar2/doorL2/door/openDoor AT 1402 : BOOL := false;
    motorCar2/doorL2/door/closeDoor AT 1403 : BOOL := false;
    motorCar2/doorL2/door/doorPosition AT 152 : REAL := 0.0;
    motorCar2/doorL2/door/length AT 153 : REAL := 1000.0;
    motorCar2/doorL2/door/doorClosedSensorLogic AT 1404 : BOOL := true;
    motorCar2/doorL2/door/doorOpenedSensorLogic AT 1405 : BOOL := true;
    motorCar2/doorL2/door/d_locking AT 1406 : BOOL := false;
    motorCar2/doorL2/door/v_d_locking AT 154 : REAL := 50.0;
    motorCar2/doorL2/door/d_doorClosedSensor AT 1407 : BOOL := false;
    motorCar2/doorL2/door/v_d_doorClosedSensor AT 1408 : BOOL := false;
    motorCar2/doorL2/door/d_doorOpenedSensor AT 1409 : BOOL := false;
    motorCar2/doorL2/door/v_d_doorOpenedSensor AT 1410 : BOOL := false;
    motorCar2/doorL3/compressedAir AT 144 : REAL := 200.0;
    motorCar2/doorL3/cmdSupply AT 1300 : BOOL := true;
    motorCar2/doorL3/sensorSupply AT 1299 : BOOL := true;
    motorCar2/doorL3/enableOpening AT 1305 : BOOL := false;
    motorCar2/doorL3/enableClosing AT 1306 : BOOL := false;
    motorCar2/doorL3/closedDoorState AT 18 : BOOL := false;
    motorCar2/doorL3/openedDoorState AT 17 : BOOL := false;
    motorCar2/doorL3/faultState AT 526 : DINT := 0;
    motorCar2/doorL3/doorPB/doorPB AT 1417 : BOOL := false;
    motorCar2/doorL3/doorPB/button AT 1421 : BOOL := false;
    motorCar2/doorL3/doorPB/_X_10 AT 1422 : BOOL := true;
    motorCar2/doorL3/doorPB/_X_11 AT 1423 : BOOL := false;
    motorCar2/doorL3/doorPB/_X_12 AT 1424 : BOOL := false;
    motorCar2/doorL3/doorLocking/lockingCmd AT 1411 : BOOL := false;
    motorCar2/doorL3/doorLocking/unlockingCmd AT 1412 : BOOL := false;
    motorCar2/doorL3/doorLocking/doorLocked AT 1415 : BOOL := false;
    motorCar2/doorL3/doorLocking/doorUnlocked AT 1416 : BOOL := false;
    motorCar2/doorL3/doorLocking/lockActive AT 1420 : BOOL := false;
    motorCar2/doorL3/doorLocking/i_rs1 AT 692 : DINT := 0;
    motorCar2/doorL3/doorLocking/d_unlockedSensor AT 1426 : BOOL := false;
    motorCar2/doorL3/doorLocking/v_d_unlockedSensor AT 1427 : BOOL := false;
    motorCar2/doorL3/doorLocking/d_lockedSensor AT 1428 : BOOL := false;
    motorCar2/doorL3/doorLocking/v_d_lockedSensor AT 1429 : BOOL := false;
    motorCar2/doorL3/doorControlPart/enableOpening AT 1305 : BOOL := false;
    motorCar2/doorL3/doorControlPart/enableClosing AT 1306 : BOOL := false;
    motorCar2/doorL3/doorControlPart/openedDoor AT 1413 : BOOL := false;
    motorCar2/doorL3/doorControlPart/closedDoor AT 1414 : BOOL := false;
    motorCar2/doorL3/doorControlPart/lockedDoor AT 1415 : BOOL := false;
    motorCar2/doorL3/doorControlPart/unlockedDoor AT 1416 : BOOL := false;
    motorCar2/doorL3/doorControlPart/openingRequest AT 1417 : BOOL := false;
    motorCar2/doorL3/doorControlPart/doorOpeningCmd AT 1418 : BOOL := false;
    motorCar2/doorL3/doorControlPart/doorClosingCmd AT 1419 : BOOL := false;
    motorCar2/doorL3/doorControlPart/doorLockingCmd AT 1411 : BOOL := false;
    motorCar2/doorL3/doorControlPart/doorUnlockingCmd AT 1412 : BOOL := false;
    motorCar2/doorL3/doorControlPart/closedDoorState AT 18 : BOOL := false;
    motorCar2/doorL3/doorControlPart/openedDoorState AT 17 : BOOL := false;
    motorCar2/doorL3/doorControlPart/faultState AT 526 : DINT := 0;
    motorCar2/doorL3/doorControlPart/_X_10 AT 1431 : BOOL := true;
    motorCar2/doorL3/doorControlPart/_X_11 AT 1432 : BOOL := false;
    motorCar2/doorL3/doorControlPart/_X_12 AT 1433 : BOOL := false;
    motorCar2/doorL3/doorControlPart/_X_13 AT 1434 : BOOL := false;
    motorCar2/doorL3/doorControlPart/_X_14 AT 1435 : BOOL := false;
    motorCar2/doorL3/doorControlPart/_X_15 AT 1436 : BOOL := false;
    motorCar2/doorL3/doorControlPart/_X_16 AT 1437 : BOOL := false;
    motorCar2/doorL3/door/compressedAir AT 144 : REAL := 200.0;
    motorCar2/doorL3/door/cmdSupply AT 1300 : BOOL := true;
    motorCar2/doorL3/door/sensorSupply AT 1299 : BOOL := true;
    motorCar2/doorL3/door/openDoorCmd AT 1418 : BOOL := false;
    motorCar2/doorL3/door/closeDoorCmd AT 1419 : BOOL := false;
    motorCar2/doorL3/door/lockActive AT 1420 : BOOL := false;
    motorCar2/doorL3/door/doorOpened AT 1413 : BOOL := false;
    motorCar2/doorL3/door/doorClosed AT 1414 : BOOL := false;
    motorCar2/doorL3/door/increment AT 155 : REAL := 0.0;
    motorCar2/doorL3/door/openDoor AT 1444 : BOOL := false;
    motorCar2/doorL3/door/closeDoor AT 1445 : BOOL := false;
    motorCar2/doorL3/door/doorPosition AT 156 : REAL := 0.0;
    motorCar2/doorL3/door/length AT 157 : REAL := 1000.0;
    motorCar2/doorL3/door/doorClosedSensorLogic AT 1446 : BOOL := true;
    motorCar2/doorL3/door/doorOpenedSensorLogic AT 1447 : BOOL := true;
    motorCar2/doorL3/door/d_locking AT 1448 : BOOL := false;
    motorCar2/doorL3/door/v_d_locking AT 158 : REAL := 50.0;
    motorCar2/doorL3/door/d_doorClosedSensor AT 1449 : BOOL := false;
    motorCar2/doorL3/door/v_d_doorClosedSensor AT 1450 : BOOL := false;
    motorCar2/doorL3/door/d_doorOpenedSensor AT 1451 : BOOL := false;
    motorCar2/doorL3/door/v_d_doorOpenedSensor AT 1452 : BOOL := false;
    motorCar2/doorR1/compressedAir AT 143 : REAL := 200.0;
    motorCar2/doorR1/cmdSupply AT 1298 : BOOL := true;
    motorCar2/doorR1/sensorSupply AT 1297 : BOOL := true;
    motorCar2/doorR1/enableOpening AT 1307 : BOOL := false;
    motorCar2/doorR1/enableClosing AT 1308 : BOOL := false;
    motorCar2/doorR1/closedDoorState AT 16 : BOOL := false;
    motorCar2/doorR1/openedDoorState AT 15 : BOOL := false;
    motorCar2/doorR1/faultState AT 525 : DINT := 0;
    motorCar2/doorR1/doorPB/doorPB AT 1459 : BOOL := false;
    motorCar2/doorR1/doorPB/button AT 1463 : BOOL := false;
    motorCar2/doorR1/doorPB/_X_10 AT 1464 : BOOL := true;
    motorCar2/doorR1/doorPB/_X_11 AT 1465 : BOOL := false;
    motorCar2/doorR1/doorPB/_X_12 AT 1466 : BOOL := false;
    motorCar2/doorR1/doorLocking/lockingCmd AT 1453 : BOOL := false;
    motorCar2/doorR1/doorLocking/unlockingCmd AT 1454 : BOOL := false;
    motorCar2/doorR1/doorLocking/doorLocked AT 1457 : BOOL := false;
    motorCar2/doorR1/doorLocking/doorUnlocked AT 1458 : BOOL := false;
    motorCar2/doorR1/doorLocking/lockActive AT 1462 : BOOL := false;
    motorCar2/doorR1/doorLocking/i_rs1 AT 695 : DINT := 0;
    motorCar2/doorR1/doorLocking/d_unlockedSensor AT 1468 : BOOL := false;
    motorCar2/doorR1/doorLocking/v_d_unlockedSensor AT 1469 : BOOL := false;
    motorCar2/doorR1/doorLocking/d_lockedSensor AT 1470 : BOOL := false;
    motorCar2/doorR1/doorLocking/v_d_lockedSensor AT 1471 : BOOL := false;
    motorCar2/doorR1/doorControlPart/enableOpening AT 1307 : BOOL := false;
    motorCar2/doorR1/doorControlPart/enableClosing AT 1308 : BOOL := false;
    motorCar2/doorR1/doorControlPart/openedDoor AT 1455 : BOOL := false;
    motorCar2/doorR1/doorControlPart/closedDoor AT 1456 : BOOL := false;
    motorCar2/doorR1/doorControlPart/lockedDoor AT 1457 : BOOL := false;
    motorCar2/doorR1/doorControlPart/unlockedDoor AT 1458 : BOOL := false;
    motorCar2/doorR1/doorControlPart/openingRequest AT 1459 : BOOL := false;
    motorCar2/doorR1/doorControlPart/doorOpeningCmd AT 1460 : BOOL := false;
    motorCar2/doorR1/doorControlPart/doorClosingCmd AT 1461 : BOOL := false;
    motorCar2/doorR1/doorControlPart/doorLockingCmd AT 1453 : BOOL := false;
    motorCar2/doorR1/doorControlPart/doorUnlockingCmd AT 1454 : BOOL := false;
    motorCar2/doorR1/doorControlPart/closedDoorState AT 16 : BOOL := false;
    motorCar2/doorR1/doorControlPart/openedDoorState AT 15 : BOOL := false;
    motorCar2/doorR1/doorControlPart/faultState AT 525 : DINT := 0;
    motorCar2/doorR1/doorControlPart/_X_10 AT 1473 : BOOL := true;
    motorCar2/doorR1/doorControlPart/_X_11 AT 1474 : BOOL := false;
    motorCar2/doorR1/doorControlPart/_X_12 AT 1475 : BOOL := false;
    motorCar2/doorR1/doorControlPart/_X_13 AT 1476 : BOOL := false;
    motorCar2/doorR1/doorControlPart/_X_14 AT 1477 : BOOL := false;
    motorCar2/doorR1/doorControlPart/_X_15 AT 1478 : BOOL := false;
    motorCar2/doorR1/doorControlPart/_X_16 AT 1479 : BOOL := false;
    motorCar2/doorR1/door/compressedAir AT 143 : REAL := 200.0;
    motorCar2/doorR1/door/cmdSupply AT 1298 : BOOL := true;
    motorCar2/doorR1/door/sensorSupply AT 1297 : BOOL := true;
    motorCar2/doorR1/door/openDoorCmd AT 1460 : BOOL := false;
    motorCar2/doorR1/door/closeDoorCmd AT 1461 : BOOL := false;
    motorCar2/doorR1/door/lockActive AT 1462 : BOOL := false;
    motorCar2/doorR1/door/doorOpened AT 1455 : BOOL := false;
    motorCar2/doorR1/door/doorClosed AT 1456 : BOOL := false;
    motorCar2/doorR1/door/increment AT 159 : REAL := 0.0;
    motorCar2/doorR1/door/openDoor AT 1486 : BOOL := false;
    motorCar2/doorR1/door/closeDoor AT 1487 : BOOL := false;
    motorCar2/doorR1/door/doorPosition AT 160 : REAL := 0.0;
    motorCar2/doorR1/door/length AT 161 : REAL := 1000.0;
    motorCar2/doorR1/door/doorClosedSensorLogic AT 1488 : BOOL := true;
    motorCar2/doorR1/door/doorOpenedSensorLogic AT 1489 : BOOL := true;
    motorCar2/doorR1/door/d_locking AT 1490 : BOOL := false;
    motorCar2/doorR1/door/v_d_locking AT 162 : REAL := 50.0;
    motorCar2/doorR1/door/d_doorClosedSensor AT 1491 : BOOL := false;
    motorCar2/doorR1/door/v_d_doorClosedSensor AT 1492 : BOOL := false;
    motorCar2/doorR1/door/d_doorOpenedSensor AT 1493 : BOOL := false;
    motorCar2/doorR1/door/v_d_doorOpenedSensor AT 1494 : BOOL := false;
    motorCar2/doorR2/compressedAir AT 142 : REAL := 200.0;
    motorCar2/doorR2/cmdSupply AT 1296 : BOOL := true;
    motorCar2/doorR2/sensorSupply AT 1295 : BOOL := true;
    motorCar2/doorR2/enableOpening AT 1307 : BOOL := false;
    motorCar2/doorR2/enableClosing AT 1308 : BOOL := false;
    motorCar2/doorR2/closedDoorState AT 14 : BOOL := false;
    motorCar2/doorR2/openedDoorState AT 13 : BOOL := false;
    motorCar2/doorR2/faultState AT 524 : DINT := 0;
    motorCar2/doorR2/doorPB/doorPB AT 1501 : BOOL := false;
    motorCar2/doorR2/doorPB/button AT 1505 : BOOL := false;
    motorCar2/doorR2/doorPB/_X_10 AT 1506 : BOOL := true;
    motorCar2/doorR2/doorPB/_X_11 AT 1507 : BOOL := false;
    motorCar2/doorR2/doorPB/_X_12 AT 1508 : BOOL := false;
    motorCar2/doorR2/doorLocking/lockingCmd AT 1495 : BOOL := false;
    motorCar2/doorR2/doorLocking/unlockingCmd AT 1496 : BOOL := false;
    motorCar2/doorR2/doorLocking/doorLocked AT 1499 : BOOL := false;
    motorCar2/doorR2/doorLocking/doorUnlocked AT 1500 : BOOL := false;
    motorCar2/doorR2/doorLocking/lockActive AT 1504 : BOOL := false;
    motorCar2/doorR2/doorLocking/i_rs1 AT 698 : DINT := 0;
    motorCar2/doorR2/doorLocking/d_unlockedSensor AT 1510 : BOOL := false;
    motorCar2/doorR2/doorLocking/v_d_unlockedSensor AT 1511 : BOOL := false;
    motorCar2/doorR2/doorLocking/d_lockedSensor AT 1512 : BOOL := false;
    motorCar2/doorR2/doorLocking/v_d_lockedSensor AT 1513 : BOOL := false;
    motorCar2/doorR2/doorControlPart/enableOpening AT 1307 : BOOL := false;
    motorCar2/doorR2/doorControlPart/enableClosing AT 1308 : BOOL := false;
    motorCar2/doorR2/doorControlPart/openedDoor AT 1497 : BOOL := false;
    motorCar2/doorR2/doorControlPart/closedDoor AT 1498 : BOOL := false;
    motorCar2/doorR2/doorControlPart/lockedDoor AT 1499 : BOOL := false;
    motorCar2/doorR2/doorControlPart/unlockedDoor AT 1500 : BOOL := false;
    motorCar2/doorR2/doorControlPart/openingRequest AT 1501 : BOOL := false;
    motorCar2/doorR2/doorControlPart/doorOpeningCmd AT 1502 : BOOL := false;
    motorCar2/doorR2/doorControlPart/doorClosingCmd AT 1503 : BOOL := false;
    motorCar2/doorR2/doorControlPart/doorLockingCmd AT 1495 : BOOL := false;
    motorCar2/doorR2/doorControlPart/doorUnlockingCmd AT 1496 : BOOL := false;
    motorCar2/doorR2/doorControlPart/closedDoorState AT 14 : BOOL := false;
    motorCar2/doorR2/doorControlPart/openedDoorState AT 13 : BOOL := false;
    motorCar2/doorR2/doorControlPart/faultState AT 524 : DINT := 0;
    motorCar2/doorR2/doorControlPart/_X_10 AT 1515 : BOOL := true;
    motorCar2/doorR2/doorControlPart/_X_11 AT 1516 : BOOL := false;
    motorCar2/doorR2/doorControlPart/_X_12 AT 1517 : BOOL := false;
    motorCar2/doorR2/doorControlPart/_X_13 AT 1518 : BOOL := false;
    motorCar2/doorR2/doorControlPart/_X_14 AT 1519 : BOOL := false;
    motorCar2/doorR2/doorControlPart/_X_15 AT 1520 : BOOL := false;
    motorCar2/doorR2/doorControlPart/_X_16 AT 1521 : BOOL := false;
    motorCar2/doorR2/door/compressedAir AT 142 : REAL := 200.0;
    motorCar2/doorR2/door/cmdSupply AT 1296 : BOOL := true;
    motorCar2/doorR2/door/sensorSupply AT 1295 : BOOL := true;
    motorCar2/doorR2/door/openDoorCmd AT 1502 : BOOL := false;
    motorCar2/doorR2/door/closeDoorCmd AT 1503 : BOOL := false;
    motorCar2/doorR2/door/lockActive AT 1504 : BOOL := false;
    motorCar2/doorR2/door/doorOpened AT 1497 : BOOL := false;
    motorCar2/doorR2/door/doorClosed AT 1498 : BOOL := false;
    motorCar2/doorR2/door/increment AT 163 : REAL := 0.0;
    motorCar2/doorR2/door/openDoor AT 1528 : BOOL := false;
    motorCar2/doorR2/door/closeDoor AT 1529 : BOOL := false;
    motorCar2/doorR2/door/doorPosition AT 164 : REAL := 0.0;
    motorCar2/doorR2/door/length AT 165 : REAL := 1000.0;
    motorCar2/doorR2/door/doorClosedSensorLogic AT 1530 : BOOL := true;
    motorCar2/doorR2/door/doorOpenedSensorLogic AT 1531 : BOOL := true;
    motorCar2/doorR2/door/d_locking AT 1532 : BOOL := false;
    motorCar2/doorR2/door/v_d_locking AT 166 : REAL := 50.0;
    motorCar2/doorR2/door/d_doorClosedSensor AT 1533 : BOOL := false;
    motorCar2/doorR2/door/v_d_doorClosedSensor AT 1534 : BOOL := false;
    motorCar2/doorR2/door/d_doorOpenedSensor AT 1535 : BOOL := false;
    motorCar2/doorR2/door/v_d_doorOpenedSensor AT 1536 : BOOL := false;
    motorCar2/doorR3/compressedAir AT 141 : REAL := 200.0;
    motorCar2/doorR3/cmdSupply AT 1294 : BOOL := true;
    motorCar2/doorR3/sensorSupply AT 1293 : BOOL := true;
    motorCar2/doorR3/enableOpening AT 1307 : BOOL := false;
    motorCar2/doorR3/enableClosing AT 1308 : BOOL := false;
    motorCar2/doorR3/closedDoorState AT 12 : BOOL := false;
    motorCar2/doorR3/openedDoorState AT 11 : BOOL := false;
    motorCar2/doorR3/faultState AT 523 : DINT := 0;
    motorCar2/doorR3/doorPB/doorPB AT 1543 : BOOL := false;
    motorCar2/doorR3/doorPB/button AT 1547 : BOOL := false;
    motorCar2/doorR3/doorPB/_X_10 AT 1548 : BOOL := true;
    motorCar2/doorR3/doorPB/_X_11 AT 1549 : BOOL := false;
    motorCar2/doorR3/doorPB/_X_12 AT 1550 : BOOL := false;
    motorCar2/doorR3/doorLocking/lockingCmd AT 1537 : BOOL := false;
    motorCar2/doorR3/doorLocking/unlockingCmd AT 1538 : BOOL := false;
    motorCar2/doorR3/doorLocking/doorLocked AT 1541 : BOOL := false;
    motorCar2/doorR3/doorLocking/doorUnlocked AT 1542 : BOOL := false;
    motorCar2/doorR3/doorLocking/lockActive AT 1546 : BOOL := false;
    motorCar2/doorR3/doorLocking/i_rs1 AT 701 : DINT := 0;
    motorCar2/doorR3/doorLocking/d_unlockedSensor AT 1552 : BOOL := false;
    motorCar2/doorR3/doorLocking/v_d_unlockedSensor AT 1553 : BOOL := false;
    motorCar2/doorR3/doorLocking/d_lockedSensor AT 1554 : BOOL := false;
    motorCar2/doorR3/doorLocking/v_d_lockedSensor AT 1555 : BOOL := false;
    motorCar2/doorR3/doorControlPart/enableOpening AT 1307 : BOOL := false;
    motorCar2/doorR3/doorControlPart/enableClosing AT 1308 : BOOL := false;
    motorCar2/doorR3/doorControlPart/openedDoor AT 1539 : BOOL := false;
    motorCar2/doorR3/doorControlPart/closedDoor AT 1540 : BOOL := false;
    motorCar2/doorR3/doorControlPart/lockedDoor AT 1541 : BOOL := false;
    motorCar2/doorR3/doorControlPart/unlockedDoor AT 1542 : BOOL := false;
    motorCar2/doorR3/doorControlPart/openingRequest AT 1543 : BOOL := false;
    motorCar2/doorR3/doorControlPart/doorOpeningCmd AT 1544 : BOOL := false;
    motorCar2/doorR3/doorControlPart/doorClosingCmd AT 1545 : BOOL := false;
    motorCar2/doorR3/doorControlPart/doorLockingCmd AT 1537 : BOOL := false;
    motorCar2/doorR3/doorControlPart/doorUnlockingCmd AT 1538 : BOOL := false;
    motorCar2/doorR3/doorControlPart/closedDoorState AT 12 : BOOL := false;
    motorCar2/doorR3/doorControlPart/openedDoorState AT 11 : BOOL := false;
    motorCar2/doorR3/doorControlPart/faultState AT 523 : DINT := 0;
    motorCar2/doorR3/doorControlPart/_X_10 AT 1557 : BOOL := true;
    motorCar2/doorR3/doorControlPart/_X_11 AT 1558 : BOOL := false;
    motorCar2/doorR3/doorControlPart/_X_12 AT 1559 : BOOL := false;
    motorCar2/doorR3/doorControlPart/_X_13 AT 1560 : BOOL := false;
    motorCar2/doorR3/doorControlPart/_X_14 AT 1561 : BOOL := false;
    motorCar2/doorR3/doorControlPart/_X_15 AT 1562 : BOOL := false;
    motorCar2/doorR3/doorControlPart/_X_16 AT 1563 : BOOL := false;
    motorCar2/doorR3/door/compressedAir AT 141 : REAL := 200.0;
    motorCar2/doorR3/door/cmdSupply AT 1294 : BOOL := true;
    motorCar2/doorR3/door/sensorSupply AT 1293 : BOOL := true;
    motorCar2/doorR3/door/openDoorCmd AT 1544 : BOOL := false;
    motorCar2/doorR3/door/closeDoorCmd AT 1545 : BOOL := false;
    motorCar2/doorR3/door/lockActive AT 1546 : BOOL := false;
    motorCar2/doorR3/door/doorOpened AT 1539 : BOOL := false;
    motorCar2/doorR3/door/doorClosed AT 1540 : BOOL := false;
    motorCar2/doorR3/door/increment AT 167 : REAL := 0.0;
    motorCar2/doorR3/door/openDoor AT 1570 : BOOL := false;
    motorCar2/doorR3/door/closeDoor AT 1571 : BOOL := false;
    motorCar2/doorR3/door/doorPosition AT 168 : REAL := 0.0;
    motorCar2/doorR3/door/length AT 169 : REAL := 1000.0;
    motorCar2/doorR3/door/doorClosedSensorLogic AT 1572 : BOOL := true;
    motorCar2/doorR3/door/doorOpenedSensorLogic AT 1573 : BOOL := true;
    motorCar2/doorR3/door/d_locking AT 1574 : BOOL := false;
    motorCar2/doorR3/door/v_d_locking AT 170 : REAL := 50.0;
    motorCar2/doorR3/door/d_doorClosedSensor AT 1575 : BOOL := false;
    motorCar2/doorR3/door/v_d_doorClosedSensor AT 1576 : BOOL := false;
    motorCar2/doorR3/door/d_doorOpenedSensor AT 1577 : BOOL := false;
    motorCar2/doorR3/door/v_d_doorOpenedSensor AT 1578 : BOOL := false;
  END_VAR
END_CONFIGURATION
